// TIA Portal V16 export
// export: Created 2021-07-14T09:31:30.8476562Z, ExportSetting WithDefaults, WithReadOnly, DisplayName Totally Integrated Automation Portal, DisplayVersion V16 Update 3, DisplayName TIA Portal Version Control Interface, DisplayVersion V16 Update 2, DisplayName TIA Portal Openness, DisplayVersion V16 Update 3, DisplayName SINAMICS Startdrive Advanced, DisplayVersion V16, DisplayName SINAMICS Startdrive G130, G150, S120, S150, SINAMICS MV, S210, DisplayVersion V16, DisplayName SINAMICS Startdrive G110M, G120, G120C, G120D, G120P, DisplayVersion V16, DisplayName STEP 7 Professional, DisplayVersion V16 Update 3, DisplayName SIMATIC Energy Suite, DisplayVersion V16, DisplayName STEP 7 Safety, DisplayVersion V16, DisplayName WinCC Advanced, DisplayVersion V16 Update 3
Screen "output"  1366x768, Number=1
  ScreenLayer 
    Rectangle "Rettangolo_1" at 237,93 size 219x72
    TextField "Casella di testo_1" at 248,129 size 82x25  Text="Variable"
    TextField "Casella di testo_2" at 248,97 size 46x25  Text="Text"
  ScreenLayer 
    Button "Pulsante_1" at 330,122 size 42x32  Mode=Text, TextOff="Set", TextOn="Text"
      on Press: SetBit(Tag := PF02D_CMD_REMOTO)
    Button "Pulsante_2" at 387,122 size 59x32  Mode=Text, TextOff="Reset", TextOn="Text"
      on Press: ResetBit(Tag := PF02D_CMD_REMOTO)
